Staubli VAL3: readENC.pgx

program readENC()
  local num l_nError
  local num l_nValue
  local string l_sValue
begin
  // Read current value from conveyor library
  resize(sCaption,1,pg:nNumOfTxtBox)
  call pg:getCaption(sCaption)
  // LatchPeriod
  call ut:_toString(enc:nLatchPeriod,"",l_sValue)
  call pg:setFieldValue(sCaption[0],l_sValue,l_nError)
  // Encoder Resolution
  call enc:getResolution(cnv:nENCRESOLUTION)
  call ut:_toString(cnv:nENCRESOLUTION,"",l_sValue)
  call pg:setFieldValue(sCaption[1],l_sValue,l_nError)
  // Display filter length
  call ut:_toString(cnv:nFirOrdre,"",l_sValue)
  call pg:setFieldValue(sCaption[2],l_sValue,l_nError)
  // display filter delay
  call ut:_toString(cnv:nFirDelay*1000,"",l_sValue)
  call pg:setFieldValue(sCaption[3],l_sValue,l_nError)
end
